Universal Robots PolyScope program: SUB_6102RXF_bak.urp

Program SUB_6102RXF_bak (installation=GD directory=/programs/GD createdIn=5.13.0 lastSavedIn=5.13.0 robotSerialNumber=20205000017)
Calibrated DH parameters: a=[-0.000157, -0.56303, -0.236706, -0.000074, -0.000109, 0]; d=[0.181705, 47.632387, 369.599619, -417.058513, 0.119878, 0.115667]; alpha=[1.570881, -0.005074, -0.001247, 1.56886, -1.570997, 0]; deltaTheta=[0, -0.405485, 5.544791, 1.143886, -0.000009, -0.000001]
InitVariablesNode
Robot Program (runOnlyOnce=false)
  SetPayload (workpieceName=k10)
  UF := Base
  SuppressedNode
    If (GP_int_in[23]>0)
      Folder ROVI_SOLVE
        If (CandCnt>0)
          Y2 := ROVI_SOLVE()
          If (Y2[0]≟10000.)
            SubPrgResult := rovi_err
            Wait Sleep waitTime=999999
      UF := Y2
  Folder M
    MoveL speed 120 mm/s, acceleration 70 mm/s^2 (useActiveTCP=false) tcp=TCP_RXF; feature=UF
      Waypoint Variable (Variable): variable(featureName=gGD_3_M_RXF)
      Wait Sleep waitTime=1
      Waypoint Variable (Variable): variable(featureName=gGD_2_M_RXF)
      Wait Sleep waitTime=1
      Popup Message (haltProgram=false message=ok? inputType=Text)
    Force Frame feature=Joint_6_name; selection=[1, 1, 1, 0, 0, 0]; wrench=[0, -10, 10, 0, 0, 0]; limitsForce=[0.005, 0.02, 0.02, 1.047198, 1.047198, 1.047198]; limitsMotion=[0.1, 0.1, 0.1, 0.349066, 0.349066, 0.349066]
      Wait Sleep waitTime=3
    Popup Message (haltProgram=false message=ok? inputType=Text)
    Force Frame feature=Joint_6_name; selection=[1, 0, 0, 0, 0, 0]; wrench=[0, 0, 0, 0, 0, 0]; limitsForce=[0.005, 0.005, 0.03, 1.047198, 1.047198, 1.047198]; limitsMotion=[0.1, 0.1, 0.1, 0.349066, 0.349066, 0.349066]
      MoveL speed 120 mm/s, acceleration 70 mm/s^2 (useActiveTCP=false) tcp=TCP_RXF; feature=UF
        Waypoint Variable (Variable): variable(featureName=gGD_1_M_RXF)
    Wait Sleep waitTime=1
    Popup Message (haltProgram=false message=ok? inputType=Text)
    Force Frame feature=Joint_6_name; selection=[1, 1, 0, 0, 0, 0]; wrench=[0, 10, 0, 0, 0, 0]; limitsForce=[0.005, 0.01, 0.15, 1.047198, 1.047198, 1.047198]; limitsMotion=[0.1, 0.1, 0.1, 0.349066, 0.349066, 0.349066]
      MoveL speed 120 mm/s, acceleration 70 mm/s^2 (useActiveTCP=false) tcp=TCP_RXF; feature=UF
        Waypoint Variable (Variable): variable(featureName=gGD_2_M_RXF)
    Wait Sleep waitTime=1
    MoveL speed 120 mm/s, acceleration 70 mm/s^2 (useActiveTCP=false) tcp=TCP_RXF; feature=UF
      Waypoint Variable (Variable): variable(featureName=gGD_3_M_RXF)
      Wait Sleep waitTime=1
  Popup Message (haltProgram=false message=ok? inputType=Text)
  Folder LM
    MoveL speed 120 mm/s, acceleration 70 mm/s^2 (useActiveTCP=false) tcp=TCP_RXF; feature=UF
      Waypoint Variable (Variable): variable(featureName=gGD_3_LM_RXF)
      Wait Sleep waitTime=1
      Waypoint Variable (Variable): variable(featureName=gGD_2_LM_RXF)
      Wait Sleep waitTime=1
      Popup Message (haltProgram=false message=ok? inputType=Text)
    Force Frame feature=Joint_6_name; selection=[1, 1, 1, 0, 0, 0]; wrench=[0, -10, 10, 0, 0, 0]; limitsForce=[0.005, 0.02, 0.005, 1.047198, 1.047198, 1.047198]; limitsMotion=[0.1, 0.1, 0.1, 0.349066, 0.349066, 0.349066]
      Wait Sleep waitTime=1
    Force Frame feature=Joint_6_name; selection=[1, 0, 0, 0, 0, 0]; wrench=[0, 0, 0, 0, 0, 0]; limitsForce=[0.005, 0.005, 0.03, 1.047198, 1.047198, 1.047198]; limitsMotion=[0.1, 0.1, 0.1, 0.349066, 0.349066, 0.349066]
      MoveL speed 120 mm/s, acceleration 70 mm/s^2 (useActiveTCP=false) tcp=TCP_RXF; feature=UF
        Waypoint Variable (Variable): variable(featureName=gGD_1_LM_RXF)
    Wait Sleep waitTime=1
    Popup Message (haltProgram=false message=ok? inputType=Text)
    Force Frame feature=Joint_6_name; selection=[1, 1, 0, 0, 0, 0]; wrench=[0, 10, 0, 0, 0, 0]; limitsForce=[0.005, 0.01, 0.15, 1.047198, 1.047198, 1.047198]; limitsMotion=[0.1, 0.1, 0.1, 0.349066, 0.349066, 0.349066]
      MoveL speed 120 mm/s, acceleration 70 mm/s^2 (useActiveTCP=false) tcp=TCP_RXF; feature=UF
        Waypoint Variable (Variable): variable(featureName=gGD_2_LM_RXF)
    Wait Sleep waitTime=1
    MoveL speed 120 mm/s, acceleration 70 mm/s^2 (useActiveTCP=false) tcp=TCP_RXF; feature=UF
      Waypoint Variable (Variable): variable(featureName=gGD_3_LM_RXF)
      Wait Sleep waitTime=1
  Popup Message (haltProgram=false message=ok? inputType=Text)
  Folder RM
    MoveL speed 120 mm/s, acceleration 70 mm/s^2 (useActiveTCP=false) tcp=TCP_RXF; feature=UF
      Waypoint Variable (Variable): variable(featureName=gGD_3_RM_RXF)
      Wait Sleep waitTime=1
      Waypoint Variable (Variable): variable(featureName=gGD_2_RM_RXF)
      Wait Sleep waitTime=1
      Popup Message (haltProgram=false message=ok? inputType=Text)
    Force Frame feature=Joint_6_name; selection=[1, 1, 1, 0, 0, 0]; wrench=[0, -10, 10, 0, 0, 0]; limitsForce=[0.005, 0.02, 0.005, 1.047198, 1.047198, 1.047198]; limitsMotion=[0.1, 0.1, 0.1, 0.349066, 0.349066, 0.349066]
      Wait Sleep waitTime=1
    Force Frame feature=Joint_6_name; selection=[1, 0, 0, 0, 0, 0]; wrench=[0, 0, 0, 0, 0, 0]; limitsForce=[0.005, 0.01, 0.15, 1.047198, 1.047198, 1.047198]; limitsMotion=[0.1, 0.1, 0.1, 0.349066, 0.349066, 0.349066]
      MoveL speed 120 mm/s, acceleration 70 mm/s^2 (useActiveTCP=false) tcp=TCP_RXF; feature=UF
        Waypoint Variable (Variable): variable(featureName=gGD_1_RM_RXF)
    Wait Sleep waitTime=1
    Popup Message (haltProgram=false message=ok? inputType=Text)
    Force Frame feature=Joint_6_name; selection=[1, 1, 0, 0, 0, 0]; wrench=[0, 10, 0, 0, 0, 0]; limitsForce=[0.005, 0.01, 0.15, 1.047198, 1.047198, 1.047198]; limitsMotion=[0.1, 0.1, 0.1, 0.349066, 0.349066, 0.349066]
      MoveL speed 120 mm/s, acceleration 70 mm/s^2 (useActiveTCP=false) tcp=TCP_RXF; feature=UF
        Waypoint Variable (Variable): variable(featureName=gGD_2_RM_RXF)
    Wait Sleep waitTime=1
    MoveL speed 120 mm/s, acceleration 70 mm/s^2 (useActiveTCP=false) tcp=TCP_RXF; feature=UF
      Waypoint Variable (Variable): variable(featureName=gGD_3_RM_RXF)
      Wait Sleep waitTime=1
  MoveL speed 120 mm/s, acceleration 70 mm/s^2 (useActiveTCP=false) tcp=TCP_1; feature=Base
    Waypoint Variable (Variable): variable(featureName=gHome_Position)
